{attribute 'GeneratedUsingTerminal: EK1110-0000-0017'}
{attribute addProperty BoxType "EK1110-0000-0017"}
{attribute addProperty Id "TcoIo.EtcSlaveTerminalBaseInfoDataAT %I*InfoData_6F19DB2B2"}
{attribute addProperty CRC "714134842"}
{attribute addProperty Size "2"}
TYPE EK1110_2A90D53A EXTENDS TcoIo.EtcSlaveTerminalBase :
STRUCT
	{attribute addProperty Name "InfoData"}
	InfoData : InfoData_6F19DB2B;
END_STRUCT
END_TYPE

(* stored: Version 1.2.0.0, ProductVersion 3.1.4024.9
   DUT EK1110_2A90D53A: Id {160d778c-c612-043a-0e38-8b80c9558750} *)
